TYPE E_ALM_PTB :
(
	TestAlarm := 1,
	MAX_E_ALM_PTB 
);
END_TYPE

(* stored: Version 1.1.0.1, ProductVersion 3.1.0.19
   DUT E_ALM_PTB: Id {185a2a6c-bbe5-44eb-8928-25bb7caef71f} *)
